{attribute addProperty BoxType "EL3318-0000-0016"}
{attribute addProperty Id "TC_ChannelAT %I*ARRAY[0..7] OF TC_Channel_897407148721090WcStateAT %I*WcState_F855686C1620InfoDataAT %I*InfoData_BC63D37F80100"}
{attribute addProperty CRC "3486888791"}
{attribute addProperty SizeInBites "968"}
{attribute addProperty SizeInBytes "121"}
TYPE EL3318_B1CC74FF :
STRUCT
	{attribute addProperty Name "TC_Channel"}
	TC_Channel : ARRAY[0..7] OF TC_Channel_89740714;
	{attribute addProperty Name "WcState"}
	WcState : WcState_F855686C;
	{attribute addProperty Name "InfoData"}
	InfoData : InfoData_BC63D37F;
END_STRUCT
END_TYPE

(* stored: Version 1.2.0.0, ProductVersion 3.1.4024.9
   DUT EL3318_B1CC74FF: Id {f43cee0d-6d68-42f3-9916-f942ea6260ba} *)
